TEXTLIST OpMode
  8 = 'CSP'
  9 = 'CSV'
  10 = 'CST'
   = ''
END_TEXTLIST

(* stored: Version 1.1.0.1, ProductVersion 3.1.4022.16
   TextList OpMode: Id {d3d0f52f-62b2-4f64-a5c5-b7f50717e2c8} *)
